Fanuc KAREL source: IO0201.KL

-- PROVISIONAL review KL for V770-1; original PC SHA256 6e992a08c22fe2ce4b005e735e7113be286d7bf1d1e110b764eb9b1796ec58fc
-- Incomplete behavior may be omitted. Consult companion uncertainty JSON. Do not deploy.
PROGRAM IO0201
%NOLOCKGROUP
-- UNRESOLVED_LOCAL_POOL 5 cells at code offset 13; source declarations unknown
-- DIRECT_LOCAL_WORD_ACCESS alone does not prove INTEGER, REAL, or BOOLEAN
BEGIN
  -- UNRESOLVED_PC offsets 0-18; opcodes 2B,2C,7B
  -- UNRESOLVED_PC offsets 23-30; opcodes 9D,23
  -- UNRESOLVED_PC offsets 35-49; opcodes 2E,22,9D,33,35
  -- UNRESOLVED_PC offsets 54-61; opcodes 9D,23
  -- UNRESOLVED_PC offsets 66-77; opcodes 2E,23
  -- UNRESOLVED_PC offsets 82-107; opcodes 27,22,22,AD,22,27,9D,31
  -- UNRESOLVED_PC offsets 112-116; opcodes 7F
  -- UNRESOLVED_PC offsets 121-125; opcodes 27,AA
  -- UNRESOLVED_PC offsets 130-134; opcodes 7F
END IO0201
